{attribute addProperty BoxType "EL4712--0000"}
{attribute addProperty Id "Ch1_ValueAT %Q*INT162"}
{attribute addProperty CRC "1318323830"}
{attribute addProperty SizeInBites "16"}
{attribute addProperty SizeInBytes "2"}
TYPE Ch1_Sample_4E940676 :
STRUCT
	{attribute addProperty Name "Ch1_Value"}
	Ch1_Value AT %Q* : INT;
END_STRUCT
END_TYPE

(* stored: Version 1.2.0.0, ProductVersion 3.1.4024.9
   DUT Ch1_Sample_4E940676: Id {3b6cac17-caed-44f6-b49c-25e2f8f68c01} *)
